FUNCTION_BLOCK CM_Merge2PartInfo (* Basic Function Block Type *)
  (* Standard: 61499-2 *)
  (* Version 0.0, 2014-11-25, 4DIAC-IDE, 4DIAC-Consortium *)
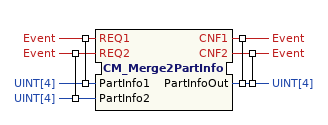
  EVENT_INPUT
    REQ1 WITH PartInfo1; (* Normal Execution Request *)
    REQ2 WITH PartInfo2;
  END_EVENT
  EVENT_OUTPUT
    CNF1 WITH PartInfoOut; (* Execution Confirmation *)
    CNF2 WITH PartInfoOut;
  END_EVENT
  VAR_INPUT
    PartInfo1 : ARRAY [0..3] OF UINT;
    PartInfo2 : ARRAY [0..3] OF UINT;
  END_VAR
  VAR_OUTPUT
    PartInfoOut : ARRAY [0..3] OF UINT;
  END_VAR
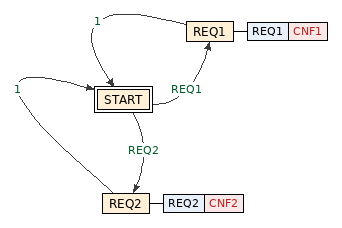
  EC_STATES
    START; (* Initial State *)
    REQ1 : REQ1 -> CNF1; (* Initialization *)
    REQ2 : REQ2 -> CNF2; (* Normal execution *)
  END_STATES
  EC_TRANSITIONS
    START TO REQ1 := REQ1;
    REQ1 TO START := 1;
    START TO REQ2 := REQ2;
    REQ2 TO START := 1;
  END_TRANSITIONS
  ALGORITHM REQ1 IN ST:
PartInfoOut[0] := PartInfo1[0];
PartInfoOut[1] := PartInfo1[1];
PartInfoOut[2] := PartInfo1[2];
PartInfoOut[3] := PartInfo1[3];
  END_ALGORITHM
  ALGORITHM REQ2 IN ST: (* Normally executed algorithm *)
PartInfoOut[0] := PartInfo2[0];
PartInfoOut[1] := PartInfo2[1];
PartInfoOut[2] := PartInfo2[2];
PartInfoOut[3] := PartInfo2[3];
  END_ALGORITHM
END_FUNCTION_BLOCK
